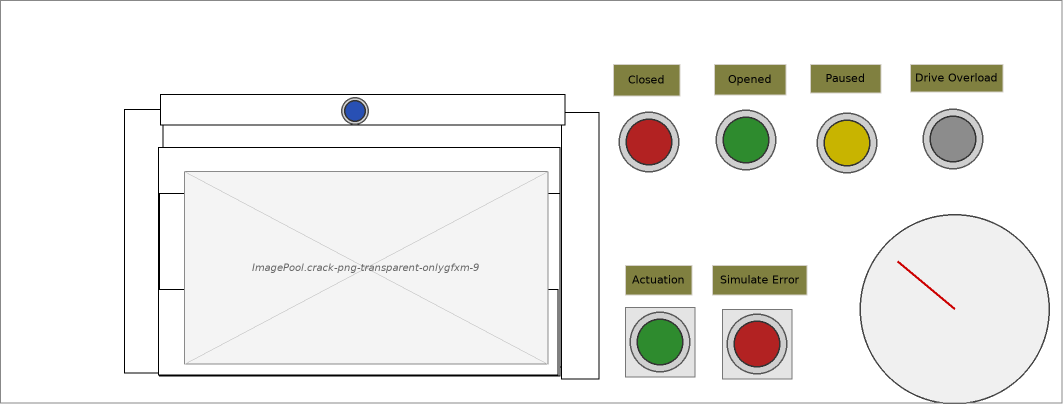
VISUALIZATION Visualization  // 1063x404
    Rectangle (161,123 402x244)
    Rectangle (124,109 39x264)
    Rectangle (561,112 38x267)
    Rectangle (160,94 405x31)
    Lamp1 (339,92 32x38), variable: GarageDoor.bMotionLight, style: Lamp-Lamp1-Blue
    Lamp1 (614,107 70x70), variable: GarageDoor.bDoorClosed, style: Lamp-Lamp1-Red
    Lamp1 (711,105 70x70), variable: GarageDoor.bDoorOpened, style: Lamp-Lamp1-Green
    Lamp1 (812,108 70x70), variable: GarageDoor.bDoorPaused, style: Lamp-Lamp1-Yellow
    Lamp1 (918,104 70x70), variable: GarageDoor.bDoorDriveOverload, style: Lamp-Lamp1-Gray
    PushSwitch (625,307 70x70), variable: GarageDoor.bActuationButton, behaviour: TAP, style: Switch-PushSwitch-Green
    PushSwitch (722,309 70x70), variable: GarageDoor.bErrorButton, behaviour: TAP, style: Switch-PushSwitch-Red
    Rectangle (161,274 399x96), invisible if: NOT GarageDoor.bTest1
    Rectangle (158,147 402x225), invisible if: NOT GarageDoor.bTest3
    Rectangle (160,205 399x166), invisible if: NOT GarageDoor.bTest2
    Rectangle (159,193 401x183), invisible if: NOT GarageDoor.bTest4
    Rectangle (158,289 400x86), invisible if: NOT GarageDoor.bTest5
    Image (184,171 364x193), invisible if: NOT GarageDoor.bErrorVis, image: ImagePool.crack-png-transparent-onlygfxm-9
    Meter360 (846,214 217x190), value: GarageDoor.fPosition, style: Meter-Meter360-Gray, scale format: %.1f, scale 0..1000
        p518627256: Actuator position
    Textfield (613,64 67x32), "Closed", colour toggle: GarageDoor.bDoorClosed
    Textfield (714,64 72x31), "Opened", colour toggle: GarageDoor.bDoorOpened
    Textfield (810,64 71x29), "Paused", colour toggle: GarageDoor.bDoorPaused
    Textfield (910,64 93x28), "Drive Overload", colour toggle: GarageDoor.bDoorDriveOverload
    Textfield (625,265 67x30), "Actuation", colour toggle: GarageDoor.bActuationButton
    Textfield (712,265 95x30), "Simulate Error", colour toggle: GarageDoor.bErrorButton
END_VISUALIZATION

(* stored: Version 1.1.0.1, ProductVersion 3.1.4024.12
   Visu Visualization: Id {76e93d4f-7cc7-4c37-872c-3d14c82ec7b2} *)
